{attribute 'qualified_only'}
VAR_GLOBAL
bStart : BOOL := FALSE; // Start button input
bStop : BOOL := FALSE; // Stop button input

bAuto : BOOL := FALSE; // Auto control mode input
bManual : BOOL := FALSE; // Manual control mode input
bOff : BOOL := FALSE; // Off mode

bJoyActive : BOOL; // Activate the joystick boolean (Top switch)
bJoyNotActive: BOOL; // Inverse logic of JoyActive
fJoyX : REAL := 0; // Variable for storing the joy value in x direction (Cylinder)
fJoyY : REAL := 0; // Variable for storing the joy value in y direction (Winch)
END_VAR

(* stored: Version 1.1.0.1, ProductVersion 3.1.4024.12
   GVL G_Virtual_Input: Id {e0169a0a-f9aa-4821-b0c4-bc7713e9c1bf} *)
